PROGRAM QueryProgram
VAR_INPUT
	sColumn:STRING(255);
END_VAR
VAR_OUTPUT
	arrRecords: ST_ProgramStruct;
	previousLine:ST_ProgramStruct;
	sSeverity: WSTRING(255);
	bError :BOOL;
	bEndOfProgram:BOOL;
	iLines: UDINT;
	bSuccess: BOOL;
	
	
END_VAR
VAR
	STProgram: ST_ProgramStruct;
	now : TIMESTRUCT;
	nowMinutes : LINT;
	fbTON: TON := ();
	fbSQLDatabase: FB_SQLDatabase(sNetID:='', tTimeout:=T#10S);
	fbPLCDBRead : FB_PLCDBRead(sNetID:='',tTimeout:=T#5S);
	fbSqlCommand : FB_SQLCommand(sNetID := '', tTimeout := T#5S);
	
	
	intTime: DINT;
	todTime: TOD;

	sCmd: STRING(255);

	dIntSqlResult: DINT;
	
	fbSQLResult: FB_SQLResult(sNetID:='', tTimeout:=T#10S);
	result: I_TcResultEvent;


	iState: INT;
	
	
	iPreviousLines: UDINT;
END_VAR




now := GVL.fbLocalSystemTime.systemTime;
nowMinutes := now.wHour*60+now.wMinute;
fbSQLDatabase:=DBConnector.fbSQLDatabase;

//State machine
CASE iState OF
0:
//IDLE
fbTON(PT := TIME#250MS);
bSuccess:=FALSE;
bEndOfProgram:=FALSE;
//Build command

sCmd :=CONCAT('SELECT * FROM [Programs] WHERE [ProgramNameID]=',LINT_TO_STRING(GVL.CurrentProgram));
sCmd :=CONCAT(sCmd,' AND [time]>');
sCmd := CONCAT(sCMD,LINT_TO_STRING(nowMinutes));
sCmd :=CONCAT(sCmd,' AND ');
sCmd := CONCAT(sCMD,sColumn);
sCmd := CONCAT(sCMD,' IS NOT NULL');
sCmd:= CONCAT(sCMD,' ORDER BY [time] ASC');
 
IF fbTON.Q=TRUE THEN
	iState:=1;
	fbTON.IN:=FALSE;
	bError := FALSE;
	
ELSE
	fbTON.IN:=TRUE;
END_IF
//Connect
1:

		IF fbSqlDatabase.bError THEN
			iState := 255;
			result := fbSqlDatabase.ipTcResultEvent;
			sSeverity := result.Text;
			 		
		ELSE
			//If sucessful, point the connection to the sql command function
			fbSqlDatabase.CreateCmd(ADR(fbSqlCommand));
			iState := 2;
		END_IF

2:
//Send the sql command
	IF fbSQLCommand.ExecuteDataReturn(ADR(sCmd), SIZEOF(sCmd), ADR(fbSqlResult)) THEN
		IF fbSQLCommand.bError THEN
			iState := 255;
			result := fbSQLCommand.ipTcResultEvent;
			sSeverity := result.Text;
			bError := TRUE;
		ELSE
			iState := 3;
			iLines:=fbSqlResult.nDataCount; 
		END_IF
	END_IF
		
3:
//Read the sql result
//If there are more than 0 lines, we're good
//If there are 0 lines we have reached the end of the program and we need to query tomorrow's program

IF iLines>0 THEN
	
	IF fbSqlResult.Read(0, 1, ADR(arrRecords), SIZEOF(arrRecords), TRUE, TRUE) THEN
		IF fbSqlResult.bError THEN
			result := fbSqlResult.ipTcResultEvent;
			sSeverity := result.Text;
			iState:=255;
			bError := TRUE;
		ELSE 
			iState:=4;
			
			result := fbSqlResult.ipTcResultEvent;
			sSeverity := result.Text;
		END_IF
	

	END_IF
	
ELSE

bEndOfProgram:=TRUE;
sCmd :=CONCAT('SELECT  *  FROM [Programs]  WHERE [ProgramNameID]=',LINT_TO_STRING(GVL.NextProgram));
sCmd :=CONCAT(sCmd,' AND ');
sCmd := CONCAT(sCMD,sColumn);
sCmd := CONCAT(sCMD,' IS NOT NULL');
sCmd := CONCAT(sCMD,' ORDER BY [time] ASC');
//Go back to state 2 and redo the query
iState:=2;

END_IF
4:
//Now build a command and query the PREVIOUS line in the program
sCmd := CONCAT('SELECT  *  FROM [Programs]  WHERE [ProgramNameID]=',LINT_TO_STRING(GVL.CurrentProgram));
sCmd := CONCAT(sCmd,' AND [time] <=');
sCmd := CONCAT(sCMD,LINT_TO_STRING(nowMinutes));
sCmd := CONCAT(sCmd,' AND ');
sCmd := CONCAT(sCMD,sColumn);
sCmd := CONCAT(sCMD,' IS NOT NULL');
sCmd := CONCAT(sCMD,' ORDER BY [time] DESC');	
	IF fbSQLCommand.ExecuteDataReturn(ADR(sCmd), SIZEOF(sCmd), ADR(fbSqlResult)) THEN
		IF fbSQLCommand.bError THEN
			iState := 255;
			result := fbSQLCommand.ipTcResultEvent;
			sSeverity := result.Text;
			bError := TRUE;
		ELSE
			iState := 5; 
			iPreviousLines:=fbSqlResult.nDataCount;
		END_IF
	END_IF

5:
//read the previous line
//If there IS a previous line then
IF iPreviousLines>0 THEN
 
	IF fbSqlResult.Read(0, 1, ADR(previousLine), SIZEOF(previousLine), TRUE, TRUE) THEN
		IF fbSqlResult.bError THEN
			result := fbSqlResult.ipTcResultEvent;
			sSeverity := result.Text;
			iState:=255;
			bError := TRUE;
		ELSE 
			//We're done go back to the beginning
			iState:=0;
			bSuccess:=TRUE; 
			result := fbSqlResult.ipTcResultEvent;
			sSeverity := result.Text;
			
		END_IF
	

	END_IF
	
//If there is NO previous line...the previous line is the next line
ELSE
	previousLine:=arrRecords;
	//We're done go back to the beginning
	iState:=0;
	bSuccess:=TRUE; 
	result := fbSqlResult.ipTcResultEvent;
	sSeverity := result.Text;
END_IF


255:
	//Record the error....I need to change this to actually record the errors
		//ADSLOGSTR(msgCtrlMask := ADSLOG_MSGTYPE_ERROR OR ADSLOG_MSGTYPE_MSGBOX, msgFmtStr := 'Oh god what have you done? %s', strArg := WSTRING_TO_STRING(result.Text));
		iState:=0;	
		bError := TRUE;
		result := fbSqlResult.ipTcResultEvent;
		sSeverity := result.Text;
	

END_CASE

END_PROGRAM

(* stored: Version 1.1.0.1, ProductVersion 3.1.4022.18
   POU QueryProgram: Id {ab1d6f67-866b-496c-bd51-28af300b2d5e}, SpecialFunc None *)
